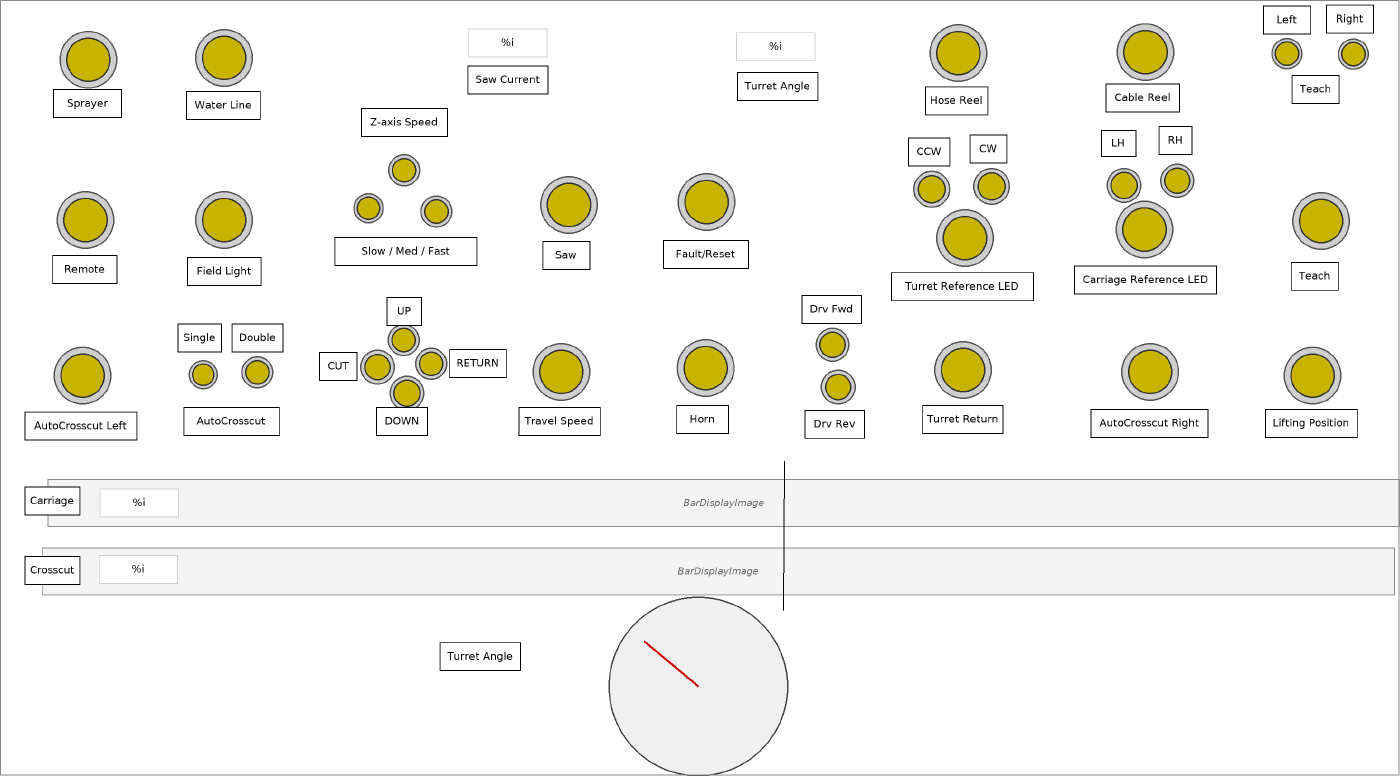
VISUALIZATION Visualization  // 1474x818
    Group (938,216 150x101)
        Lamp1 (43,0 70x70), variable: OUT_bTurretReferenceLED, style: Lamp-Lamp1-Yellow
        Rectangle (0,71 150x30), "Turret Reference LED"
    Group (1131,207 150x103)
        Lamp1 (39,0 70x70), variable: OUT_bCarriageReferenceLED, style: Lamp-Lamp1-Yellow
        Rectangle (0,73 150x30), "Carriage Reference LED"
    Lamp1 (958,177 46x45), variable: bTrtCCW, style: Lamp-Lamp1-Yellow
    Lamp1 (1020,174 48x45), variable: bTrtCW, style: Lamp-Lamp1-Yellow
    Lamp1 (1159,174 49x43), variable: bCrgLH, style: Lamp-Lamp1-Yellow
    Lamp1 (1219,170 41x41), variable: bCrgRH, style: Lamp-Lamp1-Yellow
    Rectangle (956,145 44x30), "CCW"
    Rectangle (1021,142 39x30), "CW"
    Rectangle (1159,137 37x28), "LH"
    Rectangle (1220,133 35x30), "RH"
    Lamp1 (974,21 70x70), variable: OUT_bHoseReel, style: Lamp-Lamp1-Yellow
    Lamp1 (1171,20 70x70), variable: OUT_bCableReel, style: Lamp-Lamp1-Yellow
    Lamp1 (979,355 70x70), variable: OUT_bTurretReturnLED, style: Lamp-Lamp1-Yellow
    Lamp1 (1176,357 70x70), variable: bAutoCrossCut, style: Lamp-Lamp1-Yellow
    Lamp1 (58,28 70x70), variable: OUT_bSprayer, style: Lamp-Lamp1-Yellow
    Lamp1 (201,26 70x70), variable: OUT_bWaterLine, style: Lamp-Lamp1-Yellow
    Lamp1 (55,197 70x70), variable: bRemote, style: Lamp-Lamp1-Yellow
    Lamp1 (201,197 70x70), variable: OUT_bFieldLight, style: Lamp-Lamp1-Yellow
    Lamp1 (52,361 70x70), variable: bAutoCrossCut, style: Lamp-Lamp1-Yellow
    Lamp1 (196,377 36x36), variable: bAutoCrossCutSingle, style: Lamp-Lamp1-Yellow
    Lamp1 (368,201 40x37), variable: bZAxisSlow, style: Lamp-Lamp1-Yellow
    Lamp1 (404,160 43x39), variable: bZAxisMed, style: Lamp-Lamp1-Yellow
    Lamp1 (440,203 39x40), variable: bZAxisFast, style: Lamp-Lamp1-Yellow
    Lamp1 (405,339 40x39), variable: bSawUP, style: Lamp-Lamp1-Yellow
    Lamp1 (434,364 40x39), variable: OUT_bSawRETURN, style: Lamp-Lamp1-Yellow
    Lamp1 (375,366 45x42), variable: OUT_bSawCUT, style: Lamp-Lamp1-Yellow
    Lamp1 (405,393 47x43), variable: bSawDown, style: Lamp-Lamp1-Yellow
    Lamp1 (564,181 70x70), variable: OUT_bSawONLED, style: Lamp-Lamp1-Yellow
    Lamp1 (556,357 70x70), variable: OUT_bTravelSpeedLED, style: Lamp-Lamp1-Yellow
    Lamp1 (709,178 70x70), variable: OUT_bFaultResetLED, style: Lamp-Lamp1-Yellow
    Lamp1 (708,353 70x70), variable: OUT_bHorn, style: Lamp-Lamp1-Yellow
    Lamp1 (856,343 41x41), variable: OUT_bXDriveFwd, style: Lamp-Lamp1-Yellow
    Lamp1 (857,387 51x42), variable: OUT_bXDriveRev, style: Lamp-Lamp1-Yellow
    Lamp1 (1336,37 38x39), variable: bTeachLeft, style: Lamp-Lamp1-Yellow
    Lamp1 (1402,38 46x38), variable: bTeachRight, style: Lamp-Lamp1-Yellow
    Lamp1 (1356,198 70x70), variable: OUT_bTeachLED, style: Lamp-Lamp1-Yellow
    Lamp1 (1347,361 70x70), variable: OUT_bLiftingPositionLED, style: Lamp-Lamp1-Yellow
    Rectangle (56,94 72x30), "Sprayer"
    Rectangle (196,96 78x30), "Water Line"
    Rectangle (55,269 68x30), "Remote"
    Rectangle (197,271 78x30), "Field Light"
    Rectangle (26,434 118x30), "AutoCrosscut Left"
    Rectangle (193,429 101x30), "AutoCrosscut"
    Lamp1 (251,373 40x39), variable: bAutoCrossCutDouble, style: Lamp-Lamp1-Yellow
    Rectangle (187,341 46x30), "Single"
    Rectangle (244,341 54x30), "Double"
    Rectangle (380,114 91x30), "Z-axis Speed"
    Rectangle (352,250 150x30), "Slow / Med / Fast"
    Rectangle (407,313 37x30), "UP"
    Rectangle (396,429 54x30), "DOWN"
    Rectangle (336,371 40x30), "CUT"
    Rectangle (473,368 60x30), "RETURN"
    Rectangle (571,254 50x30), "Saw"
    Rectangle (698,253 90x30), "Fault/Reset"
    Rectangle (546,429 86x30), "Travel Speed"
    Rectangle (712,427 55x30), "Horn"
    Rectangle (844,311 63x30), "Drv Fwd"
    Rectangle (847,432 63x30), "Drv Rev"
    Rectangle (971,427 85x30), "Turret Return"
    Rectangle (1148,431 124x30), "AutoCrosscut Right"
    Rectangle (974,91 66x30), "Hose Reel"
    Rectangle (1164,88 78x30), "Cable Reel"
    Rectangle (1360,79 50x30), "Teach"
    Rectangle (1359,276 50x30), "Teach"
    Rectangle (1332,431 97x30), "Lifting Position"
    Rectangle (1396,5 50x30), "Right"
    Rectangle (1330,6 50x30), "Left"
    Rectangle (776,76 85x30), "Turret Angle"
    Rectangle (492,69 85x30), "Saw Current"
    Textfield (775,34 83x30), "%i", text variable: fbTurretSSI.Out.rScaled
    Textfield (493,30 83x30), "%i", text variable: fbSawCurrent.Out.rScaled
    BarDisplayImage (50,505 1424x50), value: fbCarriagePOS.Out.rScaled, style: BarDisplayImage-Gray, scale format: %d, scale 0..41
    BarDisplayImage (44,577 1424x50), value: fbCrosscutSSI.Out.rScaled, style: BarDisplayImage-Gray, scale format: %d, scale 0..62
    Rectangle (26,513 58x30), "Carriage"
    Rectangle (26,586 58x30), "Crosscut"
    Textfield (105,515 83x30), "%i", text variable: fbCarriagePOS.Out.rScaled
    Textfield (104,585 83x30), "%i", text variable: fbCrosscutSSI.Out.rScaled
    Meter180 (552,629 366x189), value: fbTurretSSI.Out.rScaled, style: Meter-Meter180-Gray, scale format: %d, scale -90..90
        p518627256: Turret angle
    Rectangle (463,677 85x30), "Turret Angle"
    Line (825,643) (826,486)
END_VISUALIZATION

(* stored: Version 1.1.0.1, ProductVersion 3.1.4024.12
   Visu Visualization: Id {a61da31d-3d5f-407d-9655-6df1af7c1fb0} *)
